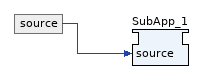
      [picture p121: application DataConnectionTestApp.Test15]
      SUBAPPLICATION SubApp_1
        VAR_INPUT
          source : ANY_INT;
        END_VAR
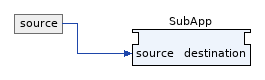
        SUBAPPLICATION SubApp
          VAR_INPUT
            source : UINT;
          END_VAR
          VAR_OUTPUT
            destination : UINT;
          END_VAR
          DATA_CONNECTIONS
            source TO destination;
          END_CONNECTIONS
        END_SUBAPPLICATION
        DATA_CONNECTIONS
          source TO SubApp.source;
        END_CONNECTIONS
      END_SUBAPPLICATION
      DATA_CONNECTIONS
        source TO SubApp_1.source;
      END_CONNECTIONS
    END_SUBAPPLICATION
    SUBAPPLICATION SubApp_21
      VAR_OUTPUT
        source : UINT;
      END_VAR
    END_SUBAPPLICATION
    SUBAPPLICATION Test17 (* event input pin with same name already exists, inwards *)
      VAR_INPUT
        source : BOOL;
      END_VAR
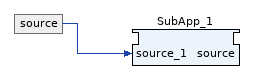
      SUBAPPLICATION SubApp_1
        VAR_INPUT
          source_1 : BOOL;
        END_VAR
        VAR_OUTPUT
          source : BOOL;
        END_VAR
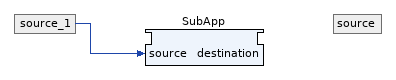
        SUBAPPLICATION SubApp
          VAR_INPUT
            source : BOOL;
          END_VAR
          VAR_OUTPUT
            destination : BOOL;
          END_VAR
          DATA_CONNECTIONS
            source TO destination;
          END_CONNECTIONS
        END_SUBAPPLICATION
        DATA_CONNECTIONS
          source_1 TO SubApp.source;
        END_CONNECTIONS
      END_SUBAPPLICATION
      DATA_CONNECTIONS
        source TO SubApp_1.source_1;
      END_CONNECTIONS
    END_SUBAPPLICATION
    SUBAPPLICATION SubApp_15
      VAR_OUTPUT
        source : BOOL;
      END_VAR
    END_SUBAPPLICATION
    SUBAPPLICATION Test19 (* incompatible data input already exists inwards, skip it *)
      VAR_INPUT
        source : INT;
      END_VAR
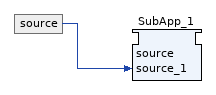
      SUBAPPLICATION SubApp_1
        VAR_INPUT
          source : UINT;
          source_1 : INT;
        END_VAR
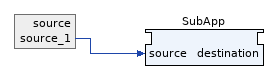
        SUBAPPLICATION SubApp
          VAR_INPUT
            source : INT;
          END_VAR
          VAR_OUTPUT
            destination : INT;
          END_VAR
          DATA_CONNECTIONS
            source TO destination;
          END_CONNECTIONS
        END_SUBAPPLICATION
        DATA_CONNECTIONS
          source_1 TO SubApp.source;
        END_CONNECTIONS
      END_SUBAPPLICATION
      DATA_CONNECTIONS
        source TO SubApp_1.source_1;
      END_CONNECTIONS
    END_SUBAPPLICATION
    SUBAPPLICATION SubApp_19
      VAR_OUTPUT
        source : INT;
      END_VAR
    END_SUBAPPLICATION
    SUBAPPLICATION Test20 (* crossing connection from FB to FB in nested subapp, data pin of same name   &#10;already exists *)
      VAR_OUTPUT
        destination : BOOL;
      END_VAR
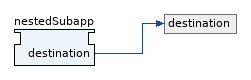
      SUBAPPLICATION nestedSubapp
        VAR_OUTPUT
          destination : BOOL;
        END_VAR
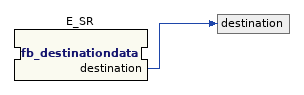
        FBS
          E_SR : fb_destinationdata;
        END_FBS
        DATA_CONNECTIONS
          E_SR.destination TO destination;
        END_CONNECTIONS
      END_SUBAPPLICATION
      DATA_CONNECTIONS
        nestedSubapp.destination TO destination;
      END_CONNECTIONS
    END_SUBAPPLICATION
    DATA_CONNECTIONS
      fb_destinationevent_1.destination TO Test4Solution.destination;
      Test5Solution.destination TO fb_destinationevent_3.source;
      Test6Solution.destination TO fb_destinationevent_5.source;
      Test7Solution.destination TO fb_destinationevent_8.source;
      Test9Solution.destination TO SubApp_9.destination_1;
      Test10Solution.destination TO SubApp_11.source;
      Test11Solution.destination TO SubApp_17.source;
      SubApp_13.source TO Test12Solution.source;
      SubApp_21.source TO Test15.source;
      SubApp_15.source TO Test17.source;
      SubApp_19.source TO Test19.source;
      Test20.destination TO fb_destinationevent_9.source;
    END_CONNECTIONS
  END_APPLICATION
END_SYSTEM
